{attribute 'linkalways'} 
{attribute 'no_explicit_call' := 'This FB is a CLASS and must be accessed using methods or properties'}
{attribute 'enable_dynamic_creation'}
FUNCTION_BLOCK FINAL ADD_LWORD EXTENDS Node
VAR
	in1 : _LWORD(0);
	in2 : _LWORD(0);
	out : _LWORD(0);
END_VAR

METHOD PUBLIC Clone : I_Node
VAR
	pNode : POINTER TO ADD_LWORD;
END_VAR
pNode := __NEW(ADD_LWORD);
Clone := pNode^;
END_METHOD

METHOD FB_init : BOOL
VAR_INPUT
	bInitRetains : BOOL; // if TRUE, the retain variables are initialized (warm start / cold start)
	bInCopyCode : BOOL;  // if TRUE, the instance afterwards gets moved into the copy code (online change)
END_VAR
AddInput('in1',THIS^.in1);
AddInput('in2',THIS^.in2);
AddOutput('out', THIS^.out);
END_METHOD

METHOD PROTECTED OnExecute
VAR
END_VAR
out.Value := in1.Value + in2.Value;
END_METHOD

END_FUNCTION_BLOCK

(* stored: Version 1.1.0.1, ProductVersion 3.1.4024.15
   POU ADD_LWORD: Id {3ea36c68-1f27-42fe-923d-f730d1c6561f}, SpecialFunc None
   Folder Constructor: Id {7b43ab29-c47a-4ef5-aa00-0e1a5905c5f6}
   Method Clone: Id {e5d3b2bd-2a07-4ecd-9e83-7fa4f30dd350}
   Method FB_init: Id {173461ab-9417-4a1e-b042-fdc767156c5d}
   Method OnExecute: Id {f80f5af4-f1e6-4272-91c2-8f2ea0bd7c5d} *)
